{attribute 'linkalways'} 
{attribute 'no_explicit_call' := 'This FB is a CLASS and must be accessed using methods or properties'}
{attribute 'enable_dynamic_creation'}
FUNCTION_BLOCK Node_F_VN_CompensateLensDistortionForPoints EXTENDS VisionNode
VAR
    ipSrcPoints : _ITcVnContainer;
    ipDestPoints : _ITcVnContainer;
    aCameraMatrix : _TcVnMatrix3x3_LREAL;
    aDistortionCoefficients : _TcVnArray4_LREAL;
    hrPrev : _HRESULT(S_OK);
	hresult : _HRESULT(S_OK);
END_VAR

METHOD PUBLIC  Clone : I_Node
VAR
	pNode : POINTER TO Node_F_VN_CompensateLensDistortionForPoints;
END_VAR
pNode := __NEW(Node_F_VN_CompensateLensDistortionForPoints);
Clone := pNode^;
END_METHOD

METHOD FB_init : BOOL
VAR_INPUT
	bInitRetains : BOOL; // if TRUE, the retain variables are initialized (warm start / cold start)
	bInCopyCode : BOOL;  // if TRUE, the instance afterwards gets moved into the copy code (online change)
END_VAR
AddInput('ipSrcPoints', ipSrcPoints);
AddInput('aCameraMatrix', aCameraMatrix);
AddInput('aDistortionCoefficients', aDistortionCoefficients);
AddInput('hrPrev', hrPrev);
AddOutput('ipDestPoints', ipDestPoints);
AddOutput('hresult', hresult);
END_METHOD

METHOD PROTECTED OnExecute
hresult.Value := F_VN_CompensateLensDistortionForPoints(
    ipSrcPoints := ipSrcPoints.Value,
	ipDestPoints := ipDestPoints.Value,
    aCameraMatrix := aCameraMatrix.Value,
    aDistortionCoefficients := aDistortionCoefficients.Value,
	hrPrev := hrPrev.Value);
END_METHOD

METHOD PUBLIC PreExecutionCheck
VAR_INPUT
	Check : I_PreExecutionChecks;
END_VAR
Check.IsTrue(ipSrcPoints.IsValid, 'ipSrcPoints must be a valid container');
Check.IsTrue((ipSrcPoints.IsType(TC_GLOBAL_CONST_LIST.ContainerType_Vector_TcVnPoint2_DINT) OR
              ipSrcPoints.IsType(TC_GLOBAL_CONST_LIST.ContainerType_Vector_TcVnPoint2_REAL)),
              'ipSrcPoints contains incorrect type');
END_METHOD

END_FUNCTION_BLOCK

(* stored: Version 1.1.0.1, ProductVersion 3.1.4026.13
   POU Node_F_VN_CompensateLensDistortionForPoints: Id {e5228544-3c16-011e-3096-e152fc0d234b}, SpecialFunc None
   Folder Constructor: Id {a6569c84-9a8c-0b60-20f3-d9df51ea657e}
   Method Clone: Id {9f9c4d83-ef8c-05d4-082f-3e2d4b4049f7}
   Method FB_init: Id {ee5cfe58-1a6e-0175-146d-4f307118331d}
   Method OnExecute: Id {9419d437-d7a7-0233-0b6e-bc230ad0262f}
   Method PreExecutionCheck: Id {d65b8b66-b9a8-03c7-14d8-bddddb2cb024} *)
